FUNCTION_BLOCK FB_FlywheelMassStorageSystem EXTENDS FB_SystemContinous
VAR_INPUT
END_VAR
VAR_OUTPUT
END_VAR
VAR
	//default parameters
	localDefaultParameters : ST_FlywheelMassStorageDefaultParameters;	

	//pumps
	stPU191DefaultParameters : ST_PumpGrundfosMagna3DefaultParameters := (tTaskCycleTime := GlobalVariables.tTaskCycleTime_MAIN, tCtrlCycleTime := GlobalVariables.tCtrlCycleTime_MAIN);
	PU191 : FB_PumpGrundfosMagna3 := (ST_DefaultParameters := stPU191DefaultParameters);;

	//valves
	stSV191DefaultParameters : ST_DiscreteValveDefaultParameters := (nFeedback := 0);
	SV191 : FB_DiscreteValve := (ST_DefaultParameters := stSV191DefaultParameters);
	
	//internal variables
	bSetStatusOn_PU191 : BOOL;
	bSetStatusOn_SV191 : BOOL;
	
	bStartTimer : BOOL;
	Timer : TON;
END_VAR

MAIN();

//use timer because valve has no feedback signal
Timer(IN := bStartTimer,
	PT := T#75S);

SV191.GetState_BI();
SV191(bSetStatusOnAutomatic := bSetStatusOn_SV191,
	bAlgorithmPermission := bAlgorithmPermission);
SV191.SetState_BO();

//pump controls return temperature
PU191.GetState_Profibus();
PU191(bSetStatusOnAutomatic := bSetStatusOn_PU191,
	bAlgorithmPermission := bAlgorithmPermission,
	fSetPointAutomatic := 70,
	nControlModeAutomatic := 0);
PU191.SetState_Profibus();

METHOD PROTECTED  CheckError : BOOL
VAR_INPUT
END_VAR
VAR_OUTPUT
	bError : BOOL;
END_VAR
bError := PU191.bError;
END_METHOD

METHOD PROTECTED  Operational : BOOL
VAR_INPUT
END_VAR
VAR_OUTPUT
	bSwitchToWorking : BOOL := FALSE;
END_VAR
bSetStatusOn_PU191 := TRUE;

IF PU191.bStatusOn THEN
	bSwitchToWorking := TRUE;
END_IF
END_METHOD

METHOD PROTECTED  RampDown : BOOL
VAR_INPUT
END_VAR
VAR_OUTPUT
	bRampDownFinished : BOOL := FALSE;
END_VAR
bSetStatusOn_PU191 := FALSE;

IF NOT PU191.bStatusOn THEN
	bSetStatusOn_SV191 := FALSE;
	bStartTimer := TRUE;
	IF Timer.Q THEN
		bStartTimer := FALSE;
		bRampDownFinished := TRUE;
	END_IF
END_IF
END_METHOD

METHOD PROTECTED  RampUp : BOOL
VAR_INPUT
END_VAR
VAR_OUTPUT
	bRampUpFinished : BOOL := FALSE;
END_VAR
bSetStatusOn_SV191 := TRUE;
bStartTimer := TRUE;

IF Timer.Q THEN
	bStartTimer := FALSE;
	bRampUpFinished := TRUE;
END_IF
END_METHOD

METHOD PROTECTED   SetSetPointLimits : BOOL
VAR_INPUT
END_VAR
aSetPointLimits[1] := localDefaultParameters.aSetPointLimitsTemperature[1];
aSetPointLimits[2] := localDefaultParameters.aSetPointLimitsTemperature[2];
END_METHOD

METHOD PROTECTED  SetState : BOOL
VAR_INPUT
END_VAR
VAR_OUTPUT
END_VAR
fOperatingPoint := PU191.fTemperatureExternal;

controlState.bStatusOn := bSetStatusOn;
setPointState.aSetPointLimits := aSetPointLimits;
setPointState.fSetPoint := fSetPoint;
setPointState.fOperatingPoint := fOperatingPoint;
setPointState.sSetPointUnit := 'degreeC';
setPointState.sOperatingPointUnit := 'degreeC';
END_METHOD

METHOD PROTECTED  Working : BOOL
VAR_INPUT
END_VAR
VAR_OUTPUT
	bSwitchToOperational : BOOL := FALSE;
END_VAR
//empty method
END_METHOD

END_FUNCTION_BLOCK

(* stored: Version 1.1.0.1, ProductVersion 3.1.4024.10
   POU FB_FlywheelMassStorageSystem: Id {1f480121-6fb9-4e01-b9b4-cf25995cf5f0}, SpecialFunc None
   Method CheckError: Id {78f9e2f0-0900-4107-96ee-83c45787b471}
   Method Operational: Id {faa262e9-eff4-4762-9e95-8afa53ca8f0b}
   Method RampDown: Id {053d2b52-e122-4bc9-b468-206bf93d4d9a}
   Method RampUp: Id {2a3903ad-bea7-46c8-a676-f0ae3f75aa8f}
   Method SetSetPointLimits: Id {cde5230d-3564-4f8f-a4cf-bb2ea6d99942}
   Method SetState: Id {d3b6743e-eab0-437e-a6a0-7ffe5a901d58}
   Method Working: Id {b6c9e5a2-9cff-41a2-bede-69a663b42e69} *)
